Omron CX-Programmer project NewProject (CX-Programmer 9.61)

# PLC NewPLC1: CP1L L

## Global symbols (name address type ; comment)
0.01 BOOL  ; Relay sinyal LM35
100.00 BOOL  ; Valve 1
100.01 BOOL  ; Valve 2
100.02 BOOL  ; Valve 1
100.03 BOOL  ; Valve 2
10.01 BOOL  ; Sistem Menyala
10.02 BOOL  ; Pengatur Delay
10.03 BOOL  ; Pompa
200 CHANNEL  ; Baca LM35
D100 CHANNEL  ; Konversi LM35
D200 CHANNEL  ; LM35 Value
T0001 BOOL  ; Delay Pengisian

## Program NewProgram1 (cyclic task 0)
Local symbols
DELAY BOOL
LT BOOL
P_off BOOL

### Section Section1

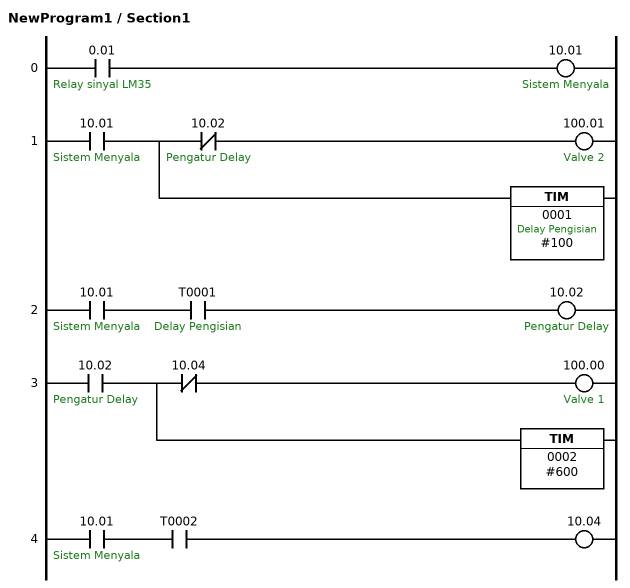
; rung 0
LD 0.01  ; Relay sinyal LM35
OUT 10.01  ; Sistem Menyala
; rung 1
LD 10.01  ; Sistem Menyala
OUT TR0
ANDNOT 10.02  ; Pengatur Delay
OUT 100.01  ; Valve 2
LD TR0
TIM 0001 #100  ; Delay Pengisian
; rung 2
LD 10.01  ; Sistem Menyala
AND T0001  ; Delay Pengisian
OUT 10.02  ; Pengatur Delay
; rung 3
LD 10.02  ; Pengatur Delay
OUT TR0
ANDNOT 10.04
OUT 100.00  ; Valve 1
LD TR0
TIM 0002 #600
; rung 4
LD 10.01  ; Sistem Menyala
AND T0002
OUT 10.04

### Section END
; rung 0
END(001)